Fanuc KAREL source: kt00895.KL

PROGRAM KT00895
%STACKSIZE=65535
%PRIORITY=65535
%NOLOCKGROUP
VAR
P1 : XYZWPREXT
P2 : XYZWPREXT
OUT : BOOLEAN
BEGIN
P1.X=1.0
P2.Y=2.0
P1.X=1.0
P2.Y=2.0
-- UNRESOLVED_PC line 12 opcodes [27 22 1C 27 9D 76 23] marker_code=80
END KT00895
